Staubli VAL3: pallet_reset.pgx

program pallet_reset(string x_sPalletName (dimensions=1))
begin
  // reset the index of the x_sPalletName
  call pallet:setPalletPos(x_sPalletName,0)
end
